# EPICS autosave request: ioc/iocBoot/iocbpmfe/auto_settings.req
file "bpmfe_settings.req",          P=$(P)
